// TIA Portal V20 export
TYPE "LKinCtrl_Picker_Kinematics_typeExternalEvents"
// stored: Access Published
   STRUCT
      kinematicsAxisSelected { ExternalAccessible := 'False'; ExternalVisible := 'False'; ExternalWritable := 'False'} : Struct
         trigger : Bool;
         axis : Int;
      END_STRUCT;
      kinematicsSelected { ExternalAccessible := 'False'; ExternalVisible := 'False'; ExternalWritable := 'False'} : Bool;
   END_STRUCT;
END_TYPE
